// TwinCAT 3 PLC project Inspection_Control
// ProgramVersion: 3.1.4026.23
// libraries:
//   CoreVision, * (Beckhoff Automation LLC)
//   Tc2_Standard, * (Beckhoff Automation GmbH)
//   Tc2_System, * (Beckhoff Automation GmbH)
//   Tc2_Utilities, * (Beckhoff Automation GmbH)
//   Tc3_PackML_V3, * (Beckhoff Automation GmbH)
//   Tc3_Vision, * (Beckhoff Automation GmbH)
//   Nestle Vanguard Base Library, * (Nestle)
//   Nestle Vanguard Wafer Inspection, * (Nestle)
// project tree:
//   GVLs/ GVL_Vision.TcGVL
//   / PlcTask.TcTTO, VisionTask.TcTTO
//   POUs/ MAIN.TcPOU, Vision.TcPOU
// real-time tasks:
//   TASK PlcTask: cycle T#10ms, priority 20, ADS port 350
//   TASK VisionTask: cycle T#50000us, priority 1, ADS port 351
//   TASK VnTask ImgAcq (FileSource1): cycle T#10ms, priority 5, ADS port 352
// I/O:
//   DEVICE Device 1 (TC3 EIP Adapter) (disabled), AmsNetId 10.201.62.134.2.1
//     Box 1 (TC EtherNet/IP Slave)

CONFIGURATION Inspection_Control
    RESOURCE PLC ON TwinCAT3
        TASK PlcTask(INTERVAL := T#10ms, PRIORITY := 20);
        TASK VisionTask(INTERVAL := T#50000us, PRIORITY := 1);
        PROGRAM MAIN WITH PlcTask : MAIN;
        PROGRAM Vision WITH VisionTask : Vision;
    END_RESOURCE
END_CONFIGURATION

// ---- GVLs/GVL_Vision.TcGVL
{attribute 'qualified_only'}
VAR_GLOBAL
	//Vision Declarations
	Camera : SimpleCamera; //Camera connection for TwinCAT vision
	WaferProcessResults : ARRAY[0..199] OF WaferResultStruct; //Results array passed by reference into the vision process
	WaferDetectionProcess : ProcessSKU(WaferResultArray := WaferProcessResults); //vision process to analyse images recieved
	ADSImageSource : ImageADSArrayReciever<5242880> := (Height := 2912, Width := 500, ChannelNumber := 1, ElementType := ETcVnElementType.TCVN_ET_UINT);
	ImageChannel : VisionChannel(Name := 'Beckhoff Camera', ImageSource := Camera, ImageProcess := WaferDetectionProcess) := (ADSImageOption := AdsImageSource); //vision channel to run the vision state machine
END_VAR

// ---- POUs/MAIN.TcPOU
PROGRAM MAIN
VAR
	// Ethernet IP inputs
	EIP_System_Ctrl : SystemControl;
	EIP_System_Ctrl_Byte AT%I* : BYTE;
	DecodeEthernetIPComms : DecodeRockwellData(Name := 'Data Decoder', SysCtrl := EIP_System_Ctrl, SysCtrlByte := EIP_System_Ctrl_Byte);
	
	// EthernetIP outputs
	EIP_System_Status : SystemStatus;
	EIP_System_Status_Bytes AT%Q* : ARRAY[0..29] OF BYTE;
	//EIP_Wafer_Results : ARRAY[0..143] OF WaferResultStruct;
	EIP_Wafer_Results_Bytes AT%Q* : ARRAY[0..719] OF BYTE;
	EncodeEthernetIPComms : EncodeBeckhoffData(Name := 'Data Encoder',
												SysSts := EIP_System_Status,
												SysStsBytes := EIP_System_Status_Bytes,
												SysWaferResultsBytes := EIP_Wafer_Results_Bytes,
												WaferResults := GVL_Vision.WaferProcessResults);
						
	//wafer detection module
	WaferVisionModule : Wafer_Inspection_Module(Name := 'Wafer Detection Module', 
												VisionChannel := GVL_Vision.ImageChannel, 
												Process := GVL_Vision.WaferDetectionProcess,
												IO_Ctrl := EIP_System_Ctrl,
												IO_Status := EIP_System_Status,
												WaferResultArray := GVL_Vision.WaferProcessResults);
	HMI : Wafer_Module_HMI('Vision Inspection',0,0);
	Init : BOOL;
END_VAR

//initialise system
//run wafer module initialisation to set up internal states
//assign module to its HJMI
IF NOT Init THEN
	Init := TRUE;
	WaferVisionModule.Initialize();
	HMI.SetModule(WaferVisionModule);
	RETURN;
END_IF

//Cyclic calls to the required objects
DecodeEthernetIPComms.CyclicLogic();
WaferVisionModule.CyclicLogic();
HMI.CyclicLogic();
EncodeEthernetIPComms.CyclicLogic();

END_PROGRAM

// ---- POUs/Vision.TcPOU
PROGRAM Vision
VAR
END_VAR

//cyclic call to the vision operations
//seperate program assigned to seperate task and run on independant core of IPC
GVL_Vision.ImageChannel.CyclicLogic();

END_PROGRAM
